FUNCTION "SM_TimeGE" : Bool
{ S7_Optimized_Access := 'FALSE' }
VERSION : 0.1
   VAR_INPUT
      value : Time;
   END_VAR

   VAR_IN_OUT
      inst : "typeSM";
   END_VAR


BEGIN
	#SM_TimeGE := (#inst.stateTime >= #value);
END_FUNCTION

